PROGRAM Data_Save
VAR
	IntervalTON     : TON;
    rtrigInterval   : R_TRIG;
    fbWritePersist  : FB_WritePersistentData;



END_VAR

END_PROGRAM

(* stored: Version 1.1.0.1, ProductVersion 3.1.4024.16
   POU Data_Save: Id {c5b6b376-ac25-4e52-bef8-9156169fe1cc}, SpecialFunc None *)
